Fanuc KAREL source: kt00090.KL

-- PROVISIONAL review KL for V1013-1; original PC SHA256 3f8120dd917dbd9ba03e6c29a81b510d18b4777065ae59d608e3df738d219f43
-- Incomplete behavior may be omitted. Consult companion uncertainty JSON. Do not deploy.
PROGRAM KT00090
%NOLOCKGROUP
VAR
  I2 : INTEGER
  OUT : REAL
-- UNRESOLVED_DECL H1 type=002017
BEGIN
  -- UNRESOLVED_PC offsets 5-19; opcodes 2E,22,9D,33,B4
  -- UNRESOLVED_PC offsets 24-35; opcodes 2E,23
  -- UNRESOLVED_PC offsets 40-63; opcodes 22,9D,33,B3,21,54,64,23
  -- UNRESOLVED_PC offsets 68-72; opcodes 7F
END KT00090
